Staubli VAL3: MotionAddon.dtx

mdesc mNomSpeed
trsf tTransformation = {rx=90}
num nXaxis
num nYaxis
num nZaxis
num nAngle
trsf trNew
num nSetAngle
num nSetXaxis
num nSetYaxis
num nSetZaxis
tool tTool = {fatherId=flange[0], ioLink=valve1}
pointRx pFbk = {fatherId=world[0]}
jointRx jFbk
num nCycleTime
num nMotState
num nMotStBit[17]
trsf trWorldExtFrc
trsf trTCPExtFrc
